TYPE ST_Message :
STRUCT
	from_slot :INT;
	to_slot	:INT;
END_STRUCT
END_TYPE

(* stored: Version 1.1.0.1, ProductVersion 3.1.4024.12
   DUT ST_Message: Id {fc87dcdc-9ee9-4991-a83c-220dba2df3d3} *)
